// TIA Portal V17 export
// export: Created 2024-01-30T08:49:13.6729507Z, ExportSetting WithDefaults, DisplayName Totally Integrated Automation Portal, DisplayVersion V17 Update 6, DisplayName TIA Portal Openness, DisplayVersion V17 Update 6, DisplayName TIA Portal Version Control Interface, DisplayVersion V17, DisplayName STEP 7 Professional, DisplayVersion V17 Update 6, DisplayName STEP 7 Safety, DisplayVersion V17 Update 6, DisplayName WinCC Advanced, DisplayVersion V17 Update 6
DATA_BLOCK "LK_G5000_DATA"   // DB16
{ S7_Optimized_Access := 'TRUE' }
VERSION : 0.1
// stored: AutoNumber true, DBAccessibleFromOPCUA true, DBAccessibleFromWebserver true, IsOnlyStoredInLoadMemory false, IsRetainMemResEnabled false, IsWriteProtectedInAS false, MemoryReserve 100
   VAR
      RS232_CTRL : Struct
         TO_LKG5000 : "UDT_LKG5000_RS232_SEND";
         FROM_LKG5000 { S7_SetPoint := 'True'} : "UDT_LKG5000_RS232_RCV";
      END_STRUCT;
      SEND_BUFF : "UDT_RS232_SEND_DATA";
      RCV_BUFF { S7_SetPoint := 'True'} : "UDT_RS232_RCV_DATA";
      RS232_Command { S7_SetPoint := 'True'} : String[11];
   END_VAR
BEGIN
END_DATA_BLOCK
